TYPE INTERNAL _BroadcastStruct :
STRUCT
	variant		: _BroadcastUnion;
	nType		: USINT;
END_STRUCT
END_TYPE

(* stored: Version 1.1.0.1
   DUT _BroadcastStruct: Id {c7a7d29f-efe7-4297-b94b-aa4eb559cb25} *)
